TYPE ST_SectorConfig :
STRUCT
	ObjectId	    : OTCID;
	PartSectorStartPosn				: LREAL;
	PartSectorEndPosn				: LREAL;
	TrackSectorStartPosn				: LREAL;
	TrackSectorEndPosn				: LREAL;
END_STRUCT
END_TYPE

(* stored: Version 1.1.0.1
   DUT ST_SectorConfig: Id {77932430-4813-013f-16b4-5b3df9147ac2} *)
